INTERFACE I_DT EXTENDS I_Datatype

PROPERTY PUBLIC Value : REFERENCE TO DT
GET
END_GET
END_PROPERTY

END_INTERFACE

(* stored: Version 1.1.0.1, ProductVersion 3.1.4024.15
   Itf I_DT: Id {5814b887-6bf9-09a4-1f72-dbd5a3602ee0}
   Property Value: Id {b75375bf-82de-05d9-3869-6048998d6667}
   Get Get: Id {7ef68876-36b1-086d-2a19-f3461b9a55ee} *)
